% RSLogix 500 project LVD190607.RSS, saved by version 11.00.00.00 %
PROJECT "LINL0619"    % processor: MicroLogix 1400 %

PROGRAM FILES
  LAD 2 "MAIN"  60 rungs  % Main Program Routine %
  LAD 3 "TEST"  7 rungs
  LAD 4 "ENABLES"  16 rungs
  LAD 6 "FEED"  11 rungs  % normal %
  LAD 8 "SPEEDS"  12 rungs
  LAD 20 "HSC BOT"  5 rungs
  LAD 22 "HSC TOP"  5 rungs
  LAD 30 "1 MS STI"  23 rungs  % high speed %
  LAD 40 "SHIFT BOT"  8 rungs
  LAD 42 "SHIFT TOP"  10 rungs
  LAD 50 "BOTOPTIC"  3 rungs
  LAD 52 "BOTOPTMES"  7 rungs
  LAD 80 "XFER"  3 rungs
  LAD 90 "TOPOPTIC"  10 rungs
  LAD 91 "TOPOPVERT"  13 rungs
  LAD 92 "TOPOPREAL"  19 rungs
  LAD 93 "TOPOPTEST"  8 rungs
  LAD 94 "TOPOPRANGE"  6 rungs
  LAD 95 "TOPOPOKAY"  6 rungs
  LAD 96 "TESTINJECT"  10 rungs
  LAD 100 "I5"  22 rungs
  LAD 101 "I5 RESULT"  7 rungs
  LAD 102 "I5 PASS"  6 rungs
  LAD 103 "I5 FAIL"  4 rungs
  LAD 104 "I5 ACQ"  9 rungs
  LAD 105 "I5 TESTER"  5 rungs
  LAD 106 "I5 TRIG"  5 rungs
  LAD 107 "I5 FIFOSET"  9 rungs
  LAD 108 "I5 FIFOGET"  8 rungs
  LAD 109 "I5 DATA"  3 rungs
  LAD 110 "I5 FAULT"  9 rungs
  LAD 111 "I5 FIX1"  5 rungs
  LAD 112 "I5 FIX2"  3 rungs
  LAD 120 "I6"  21 rungs
  LAD 121 "I6 RESULT"  7 rungs
  LAD 122 "I6 PASS"  5 rungs
  LAD 123 "I6 FAIL"  3 rungs
  LAD 124 "I6 ACQ"  8 rungs
  LAD 125 "I6 TESTER"  5 rungs
  LAD 126 "I6 TRIG"  5 rungs
  LAD 127 "I6 FIFOSET"  9 rungs
  LAD 128 "I6 FIFOGET"  8 rungs
  LAD 129 "I6 DATA"  3 rungs
  LAD 130 "I6 FAULT"  9 rungs
  LAD 131 "I6 FIX1"  5 rungs
  LAD 132 "I6 FIX2"  3 rungs
  LAD 140 "I7"  21 rungs
  LAD 141 "I7 RESULT"  7 rungs
  LAD 142 "I7 PASS"  6 rungs
  LAD 143 "I7 FAIL"  4 rungs
  LAD 144 "I7 ACQ"  9 rungs
  LAD 145 "I7 TESTER"  5 rungs
  LAD 146 "I7 TRIG"  5 rungs
  LAD 147 "I7 FIFOSET"  9 rungs
  LAD 148 "I7 FIFOGET"  8 rungs
  LAD 149 "I7 DATA"  3 rungs
  LAD 150 "I7 FAULT"  9 rungs
  LAD 151 "I7 FIX1"  5 rungs
  LAD 152 "I7 FIX2"  3 rungs
  LAD 160 "I8"  22 rungs
  LAD 161 "I8 RESULT"  7 rungs
  LAD 162 "I8 PASS"  6 rungs
  LAD 163 "I8 FAIL"  4 rungs
  LAD 164 "I8 ACQ"  9 rungs
  LAD 165 "I8 TESTER"  5 rungs
  LAD 166 "I8 TRIG"  5 rungs
  LAD 167 "I8 FIFOSET"  9 rungs
  LAD 168 "I8 FIFOGET"  8 rungs
  LAD 169 "I8 DATA"  3 rungs
  LAD 170 "I8 FAULT"  9 rungs
  LAD 171 "I8 FIX1"  5 rungs
  LAD 172 "I8 FIX2"  3 rungs
  LAD 200 "PASS BLOW"  15 rungs
  LAD 213 "TESTTRIG1"  4 rungs
  LAD 214 "TESTTRIG5"  4 rungs
  LAD 215 "TESTTRIG6"  4 rungs
  LAD 216 "TESTTRIG7"  4 rungs
  LAD 217 "TESTTRIG8"  4 rungs
  LAD 219 "PACKAGER"  28 rungs  % normal %
  LAD 220 "NO PACKAGE"  8 rungs
  LAD 222 "RATE1"  9 rungs
  LAD 223 "RATE2"  6 rungs
  LAD 224 "RESET RATE"  6 rungs
  LAD 240 "NP STOP"  8 rungs
  LAD 246 "SPEED BOT"  8 rungs  % high speed %
  LAD 248 "SPEED TOP"  8 rungs  % high speed %
  LAD 250 "P BOT"  7 rungs  % high speed %
  LAD 252 "P TOP"  7 rungs  % high speed %
  LAD 254 "TOTALCOUNT"  4 rungs
  LAD 255 "SAVED"  4 rungs

DATA FILES
  O0 OUTPUT  11 elements
  I1 INPUT  11 elements
  S2 STATUS  66 elements
  B3 BINARY  14 elements
  T4 TIMER  45 elements
  C5 COUNTER  1 elements
  R6 CONTROL  30 elements
  N7 INTEGER  200 elements
  F8 FLOAT  100 elements
  B12 HMI_BINARY  22 elements  % general use with hmi to avoid additional reads %
  L13  COUNTS  256 elements
  F14 HMI_FLOATS  100 elements
  N15 HMI_INTS  100 elements
  L16 HMI_LONGS  100 elements
  L19 RATE DATA  50 elements
  L20 I7TIMEFIFO  50 elements
  L21 I7POSFIFO  50 elements
  L22 I8TIMEFIFO  50 elements
  L23 I8POSFIFO  50 elements
  L30 INS5TIME  50 elements
  L31 INS5POS  50 elements
  L32 INS6TIME  50 elements
  L33 INS6POS  50 elements
  B34 BOT NG  128 elements
  B35 TOP NG  128 elements
  B36 BOTGOOD  128 elements
  B37 TOPGOOD1  128 elements
  B38 EX1 TEST  128 elements
  B39 TOPGOOD2  128 elements
  B40 EX2 TEST  128 elements
  N184 TEST INTS  50 elements
  L192 SPD OFFSET  50 elements
  B196 CTRL BITS  50 elements
  L199 USED  36 elements

LADDER 2 "MAIN"    % Main Program Routine %
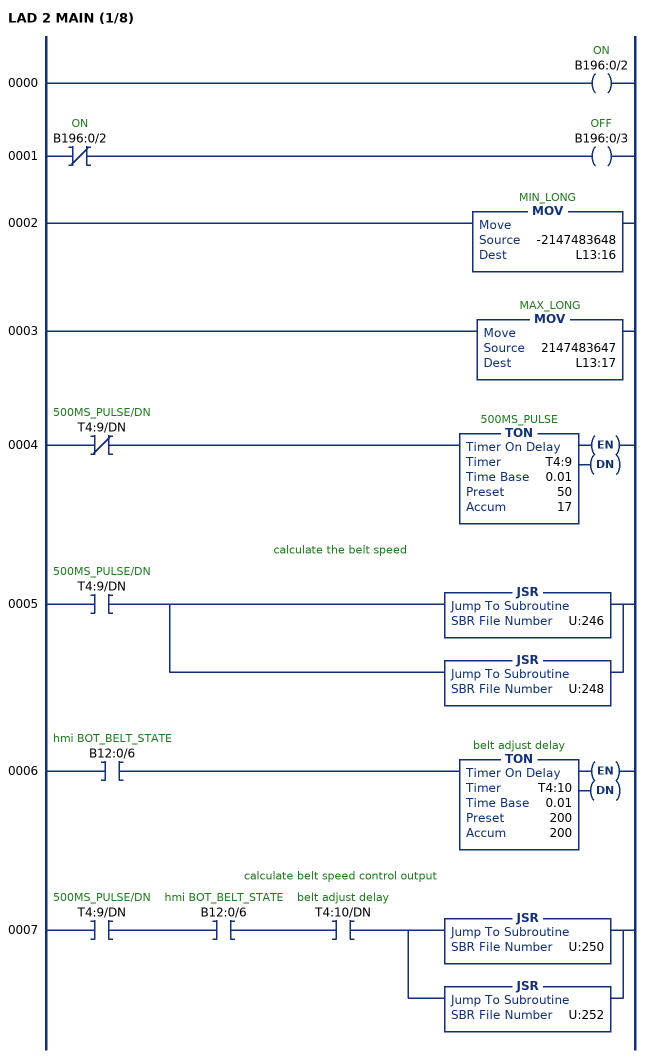
% Rung: 0 %
SOR OTE B196:0/2 EOR
%   B196:0/2  ON %
% Rung: 1 %
SOR XIO B196:0/2 OTE B196:0/3 EOR
%   B196:0/2  ON %
%   B196:0/3  OFF %
% Rung: 2 %
SOR MOV -2147483648 L13:16 EOR
%   L13:16  MIN_LONG %
% Rung: 3 %
SOR MOV 2147483647 L13:17 EOR
%   L13:17  MAX_LONG %
% Rung: 4 %
SOR XIO T4:9/DN TON T4:9 0.01 50 17 EOR
%   T4:9  500MS_PULSE %
% Rung: 5 %
% calculate the belt speed %
SOR XIC T4:9/DN BST JSR U:246 NXB JSR U:248 BND EOR
%   T4:9  500MS_PULSE %
% Rung: 6 %
SOR XIC B12:0/6 TON T4:10 0.01 200 200 EOR
%   B12:0/6  BOT_BELT_STATE  "hmi" %
%   T4:10  "belt adjust delay" %
% Rung: 7 %
% calculate belt speed control output %
SOR XIC T4:9/DN XIC B12:0/6 XIC T4:10/DN BST JSR U:250 NXB JSR U:252 BND EOR
%   T4:9  500MS_PULSE %
%   B12:0/6  BOT_BELT_STATE  "hmi" %
%   T4:10  "belt adjust delay" %

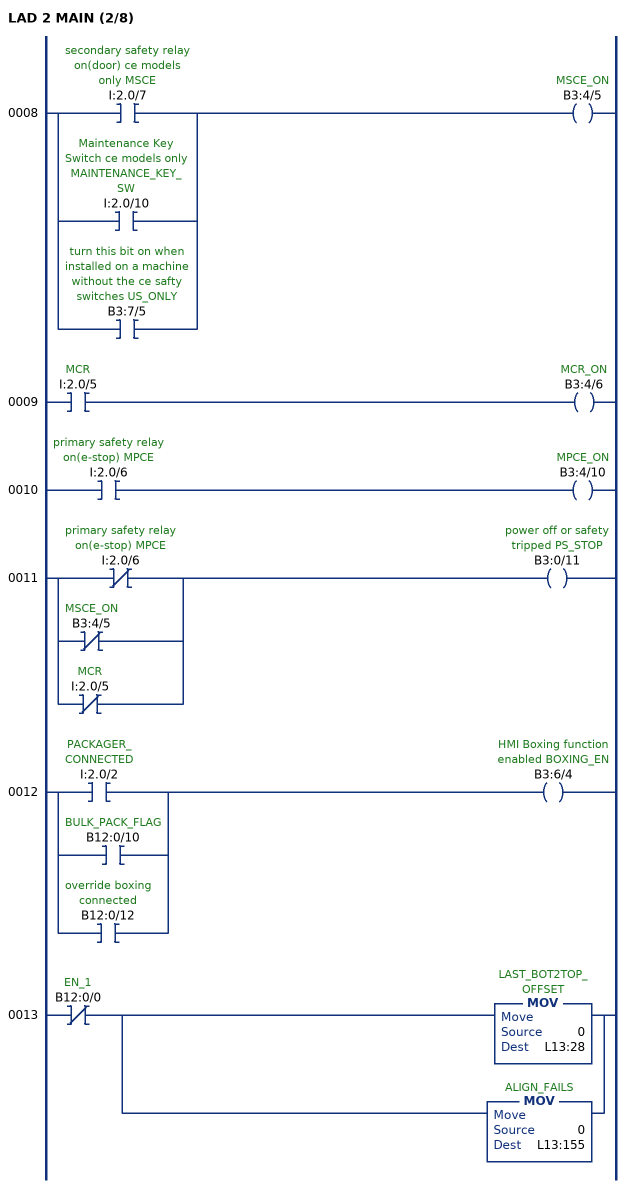
% Rung: 8 %
SOR BST XIC I:2.0/7 NXB XIC I:2.0/10 NXB XIC B3:7/5 BND OTE B3:4/5 EOR
%   I:2.0/7  MSCE  "secondary safety relay on(door) ce models only" %
%   I:2.0/10  MAINTENANCE_KEY_SW  "Maintenance Key Switch ce models only" %
%   B3:7/5  US_ONLY  "turn this bit on when installed on a machine without the ce safty switches" %
%   B3:4/5  MSCE_ON %
% Rung: 9 %
SOR XIC I:2.0/5 OTE B3:4/6 EOR
%   I:2.0/5  MCR %
%   B3:4/6  MCR_ON %
% Rung: 10 %
SOR XIC I:2.0/6 OTE B3:4/10 EOR
%   I:2.0/6  MPCE  "primary safety relay on(e-stop)" %
%   B3:4/10  MPCE_ON %
% Rung: 11 %
SOR BST XIO I:2.0/6 NXB XIO B3:4/5 NXB XIO I:2.0/5 BND OTE B3:0/11 EOR
%   I:2.0/6  MPCE  "primary safety relay on(e-stop)" %
%   B3:4/5  MSCE_ON %
%   I:2.0/5  MCR %
%   B3:0/11  PS_STOP  "power off or safety tripped" %
% Rung: 12 %
SOR BST XIC I:2.0/2 NXB XIC B12:0/10 NXB XIC B12:0/12 BND OTE B3:6/4 EOR
%   I:2.0/2  PACKAGER_CONNECTED %
%   B12:0/10  BULK_PACK_FLAG %
%   B12:0/12  "override boxing connected" %
%   B3:6/4  BOXING_EN  "HMI Boxing function enabled" %
% Rung: 13 %
SOR XIO B12:0/0 BST MOV 0 L13:28 NXB MOV 0 L13:155 BND EOR
%   B12:0/0  EN_1 %
%   L13:28  LAST_BOT2TOP_OFFSET %
%   L13:155  ALIGN_FAILS %

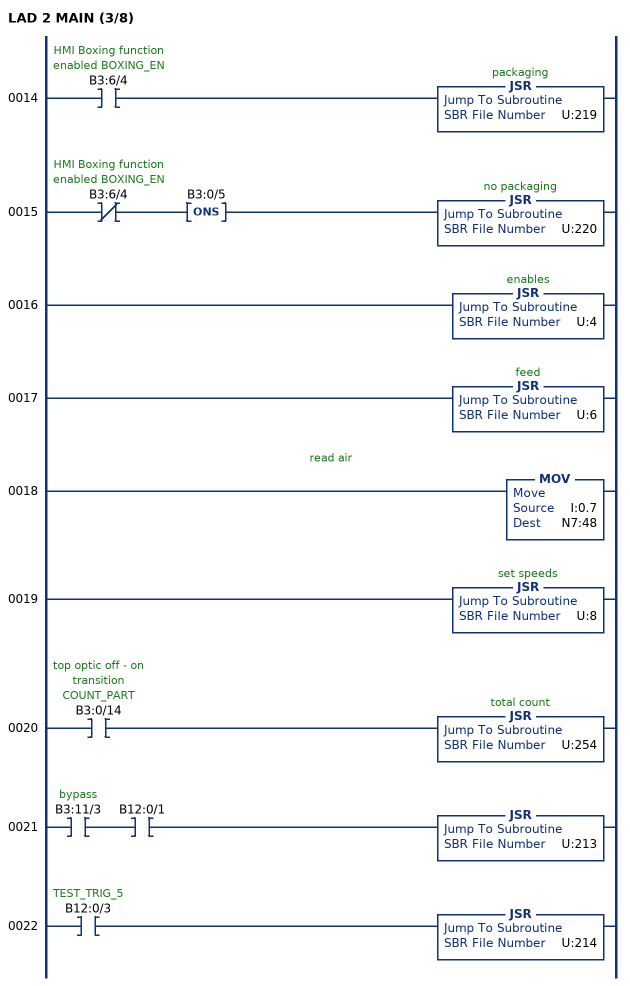
% Rung: 14 %
SOR XIC B3:6/4 JSR U:219 EOR
%   B3:6/4  BOXING_EN  "HMI Boxing function enabled" %
%   U:219  "packaging" %
% Rung: 15 %
SOR XIO B3:6/4 ONS B3:0/5 JSR U:220 EOR
%   B3:6/4  BOXING_EN  "HMI Boxing function enabled" %
%   U:220  "no packaging" %
% Rung: 16 %
SOR JSR U:4 EOR
%   U:4  "enables" %
% Rung: 17 %
SOR JSR U:6 EOR
%   U:6  "feed" %
% Rung: 18 %
% read air %
SOR MOV I:0.7 N7:48 EOR
%   I:0.7  "Air Presure Sensor Input Signal" %
% Rung: 19 %
SOR JSR U:8 EOR
%   U:8  "set speeds" %
% Rung: 20 %
SOR XIC B3:0/14 JSR U:254 EOR
%   B3:0/14  COUNT_PART  "top optic off - on transition" %
%   U:254  "total count" %
% Rung: 21 %
SOR XIC B3:11/3 XIC B12:0/1 JSR U:213 EOR
%   B3:11/3  "bypass" %
% Rung: 22 %
SOR XIC B12:0/3 JSR U:214 EOR
%   B12:0/3  TEST_TRIG_5 %

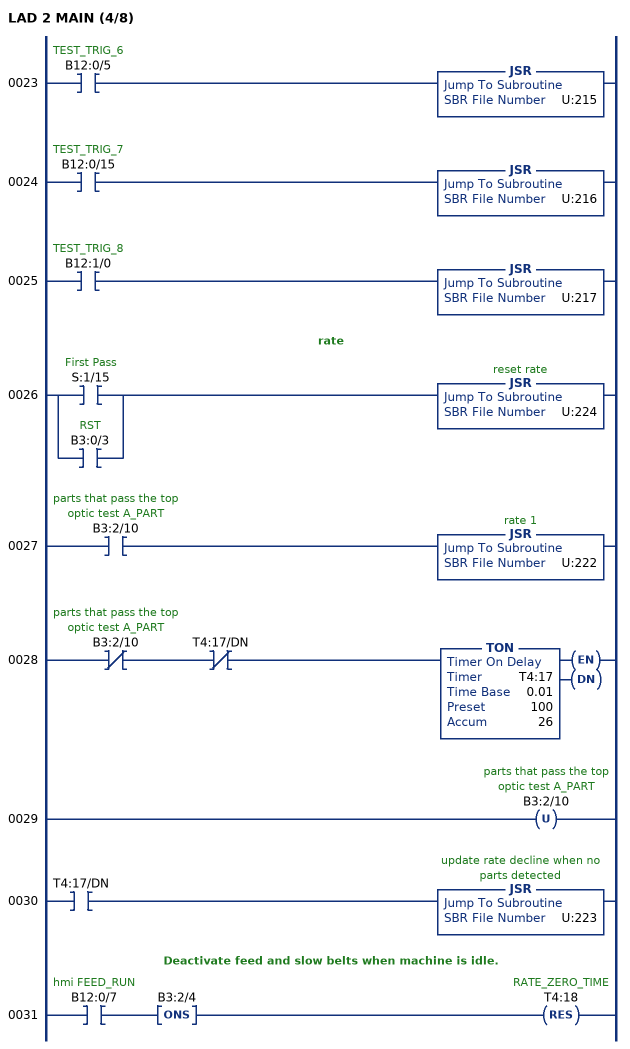
% Rung: 23 %
SOR XIC B12:0/5 JSR U:215 EOR
%   B12:0/5  TEST_TRIG_6 %
% Rung: 24 %
SOR XIC B12:0/15 JSR U:216 EOR
%   B12:0/15  TEST_TRIG_7 %
% Rung: 25 %
SOR XIC B12:1/0 JSR U:217 EOR
%   B12:1/0  TEST_TRIG_8 %
% Rung: 26 %
% TITLE: rate %
SOR BST XIC S:1/15 NXB XIC B3:0/3 BND JSR U:224 EOR
%   S:1/15  "First Pass" %
%   B3:0/3  RST %
%   U:224  "reset rate" %
% Rung: 27 %
SOR XIC B3:2/10 JSR U:222 EOR
%   B3:2/10  A_PART  "parts that pass the top optic test" %
%   U:222  "rate 1" %
% Rung: 28 %
SOR XIO B3:2/10 XIO T4:17/DN TON T4:17 0.01 100 26 EOR
%   B3:2/10  A_PART  "parts that pass the top optic test" %
% Rung: 29 %
SOR OTU B3:2/10 EOR
%   B3:2/10  A_PART  "parts that pass the top optic test" %
% Rung: 30 %
SOR XIC T4:17/DN JSR U:223 EOR
%   U:223  "update rate decline when no parts detected" %
% Rung: 31 %
% TITLE: Deactivate feed and slow belts when machine is idle. %
SOR XIC B12:0/7 ONS B3:2/4 RES T4:18 EOR
%   B12:0/7  FEED_RUN  "hmi" %
%   T4:18  RATE_ZERO_TIME %

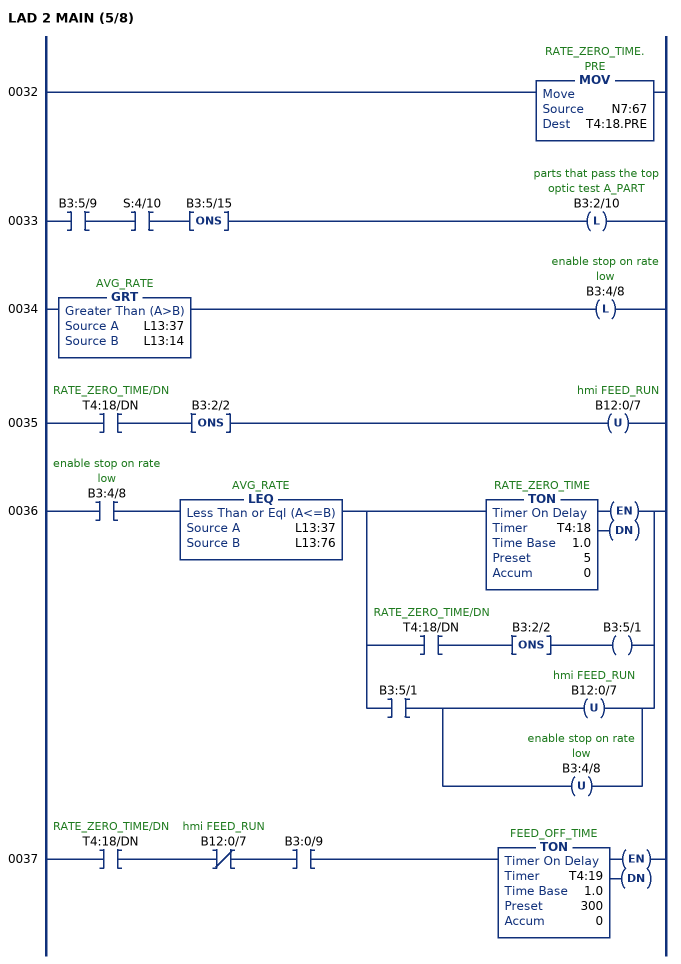
% Rung: 32 %
SOR MOV N7:67 T4:18.PRE EOR
%   N7:67  "empty bowl or jam bowl run time" %
%   T4:18  RATE_ZERO_TIME %
% Rung: 33 %
SOR XIC B3:5/9 XIC S:4/10 ONS B3:5/15 OTL B3:2/10 EOR
%   B3:2/10  A_PART  "parts that pass the top optic test" %
% Rung: 34 %
SOR GRT L13:37 L13:14 OTL B3:4/8 EOR
%   L13:37  AVG_RATE %
%   B3:4/8  "enable stop on rate low" %
% Rung: 35 %
SOR XIC T4:18/DN ONS B3:2/2 OTU B12:0/7 EOR
%   T4:18  RATE_ZERO_TIME %
%   B12:0/7  FEED_RUN  "hmi" %
% Rung: 36 %
SOR XIC B3:4/8 LEQ L13:37 L13:76 BST TON T4:18 1.0 5 0 NXB XIC T4:18/DN ONS B3:2/2 OTE B3:5/1 NXB XIC B3:5/1 BST OTU B12:0/7 NXB OTU B3:4/8 BND BND EOR
%   B3:4/8  "enable stop on rate low" %
%   L13:37  AVG_RATE %
%   T4:18  RATE_ZERO_TIME %
%   B12:0/7  FEED_RUN  "hmi" %
% Rung: 37 %
SOR XIC T4:18/DN XIO B12:0/7 XIC B3:0/9 TON T4:19 1.0 300 0 EOR
%   T4:18  RATE_ZERO_TIME %
%   B12:0/7  FEED_RUN  "hmi" %
%   T4:19  FEED_OFF_TIME %

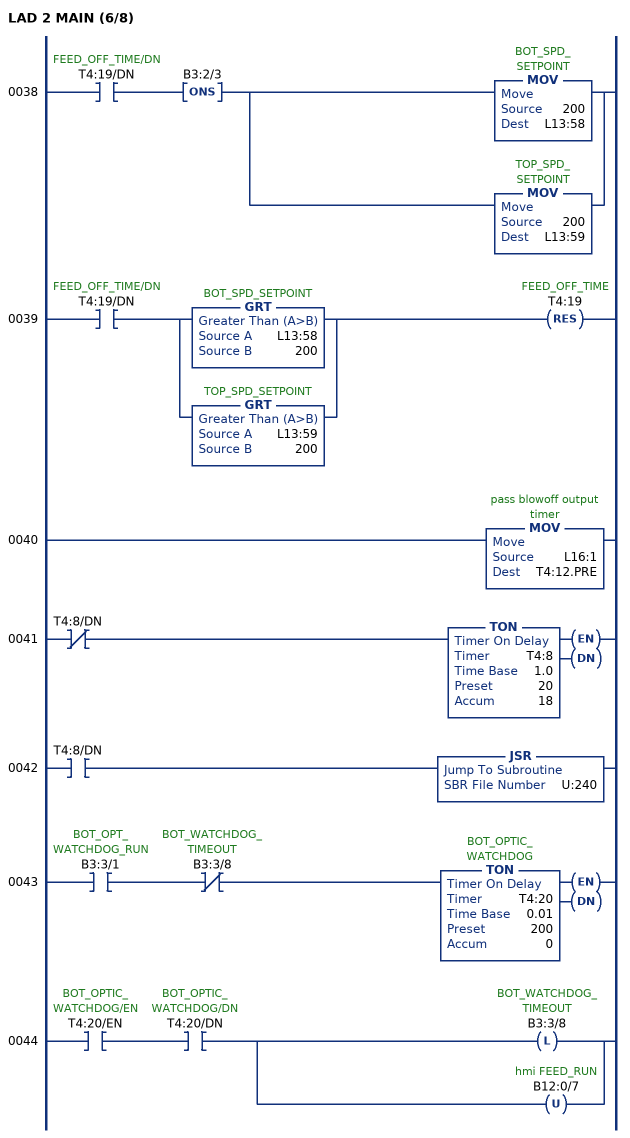
% Rung: 38 %
SOR XIC T4:19/DN ONS B3:2/3 BST MOV 200 L13:58 NXB MOV 200 L13:59 BND EOR
%   T4:19  FEED_OFF_TIME %
%   L13:58  BOT_SPD_SETPOINT %
%   L13:59  TOP_SPD_SETPOINT %
% Rung: 39 %
SOR XIC T4:19/DN BST GRT L13:58 200 NXB GRT L13:59 200 BND RES T4:19 EOR
%   T4:19  FEED_OFF_TIME %
%   L13:58  BOT_SPD_SETPOINT %
%   L13:59  TOP_SPD_SETPOINT %
% Rung: 40 %
SOR MOV L16:1 T4:12.PRE EOR
%   L16:1  BLOW_TIME %
%   T4:12  "pass blowoff output timer" %
% Rung: 41 %
SOR XIO T4:8/DN TON T4:8 1.0 20 18 EOR
% Rung: 42 %
SOR XIC T4:8/DN JSR U:240 EOR
% Rung: 43 %
SOR XIC B3:3/1 XIO B3:3/8 TON T4:20 0.01 200 0 EOR
%   B3:3/1  BOT_OPT_WATCHDOG_RUN %
%   B3:3/8  BOT_WATCHDOG_TIMEOUT %
%   T4:20  BOT_OPTIC_WATCHDOG %
% Rung: 44 %
SOR XIC T4:20/EN XIC T4:20/DN BST OTL B3:3/8 NXB OTU B12:0/7 BND EOR
%   T4:20  BOT_OPTIC_WATCHDOG %
%   B3:3/8  BOT_WATCHDOG_TIMEOUT %
%   B12:0/7  FEED_RUN  "hmi" %

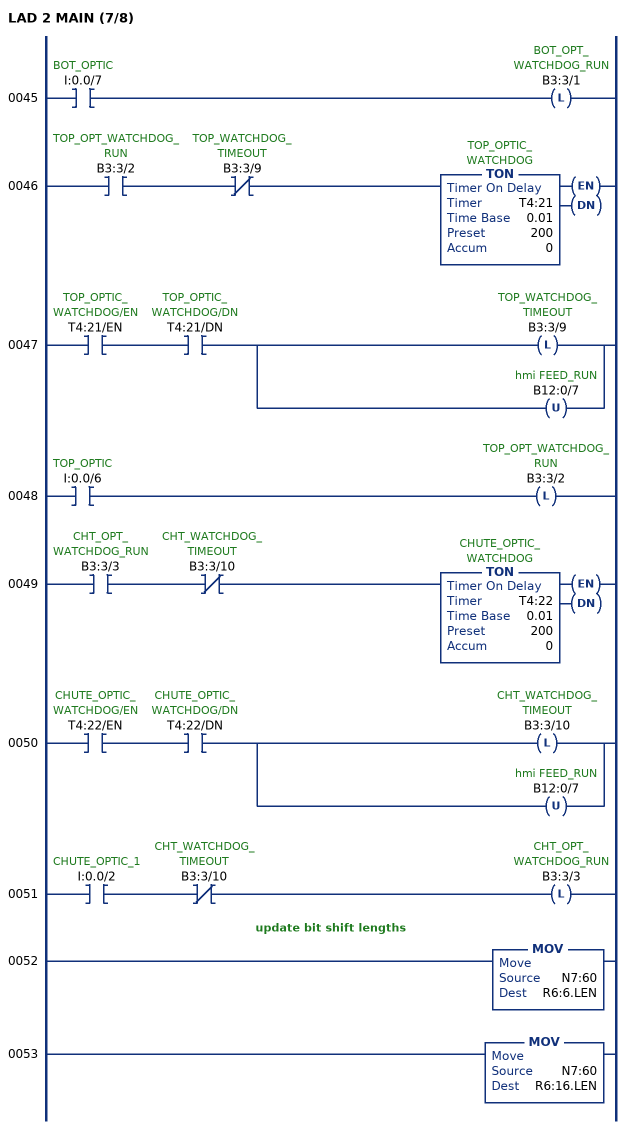
% Rung: 45 %
SOR XIC I:0.0/7 OTL B3:3/1 EOR
%   I:0.0/7  BOT_OPTIC %
%   B3:3/1  BOT_OPT_WATCHDOG_RUN %
% Rung: 46 %
SOR XIC B3:3/2 XIO B3:3/9 TON T4:21 0.01 200 0 EOR
%   B3:3/2  TOP_OPT_WATCHDOG_RUN %
%   B3:3/9  TOP_WATCHDOG_TIMEOUT %
%   T4:21  TOP_OPTIC_WATCHDOG %
% Rung: 47 %
SOR XIC T4:21/EN XIC T4:21/DN BST OTL B3:3/9 NXB OTU B12:0/7 BND EOR
%   T4:21  TOP_OPTIC_WATCHDOG %
%   B3:3/9  TOP_WATCHDOG_TIMEOUT %
%   B12:0/7  FEED_RUN  "hmi" %
% Rung: 48 %
SOR XIC I:0.0/6 OTL B3:3/2 EOR
%   I:0.0/6  TOP_OPTIC %
%   B3:3/2  TOP_OPT_WATCHDOG_RUN %
% Rung: 49 %
SOR XIC B3:3/3 XIO B3:3/10 TON T4:22 0.01 200 0 EOR
%   B3:3/3  CHT_OPT_WATCHDOG_RUN %
%   B3:3/10  CHT_WATCHDOG_TIMEOUT %
%   T4:22  CHUTE_OPTIC_WATCHDOG %
% Rung: 50 %
SOR XIC T4:22/EN XIC T4:22/DN BST OTL B3:3/10 NXB OTU B12:0/7 BND EOR
%   T4:22  CHUTE_OPTIC_WATCHDOG %
%   B3:3/10  CHT_WATCHDOG_TIMEOUT %
%   B12:0/7  FEED_RUN  "hmi" %
% Rung: 51 %
SOR XIC I:0.0/2 XIO B3:3/10 OTL B3:3/3 EOR
%   I:0.0/2  CHUTE_OPTIC_1 %
%   B3:3/10  CHT_WATCHDOG_TIMEOUT %
%   B3:3/3  CHT_OPT_WATCHDOG_RUN %
% Rung: 52 %
% TITLE: update bit shift lengths %
SOR MOV N7:60 R6:6.LEN EOR
% Rung: 53 %
SOR MOV N7:60 R6:16.LEN EOR

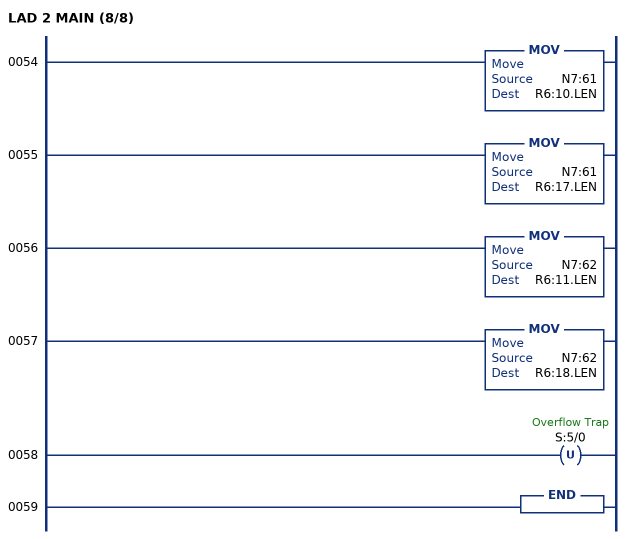
% Rung: 54 %
SOR MOV N7:61 R6:10.LEN EOR
% Rung: 55 %
SOR MOV N7:61 R6:17.LEN EOR
% Rung: 56 %
SOR MOV N7:62 R6:11.LEN EOR
% Rung: 57 %
SOR MOV N7:62 R6:18.LEN EOR
% Rung: 58 %
SOR OTU S:5/0 EOR
%   S:5/0  "Overflow Trap" %
% Rung: 59 %
SOR END EOR

LADDER 3 "TEST"
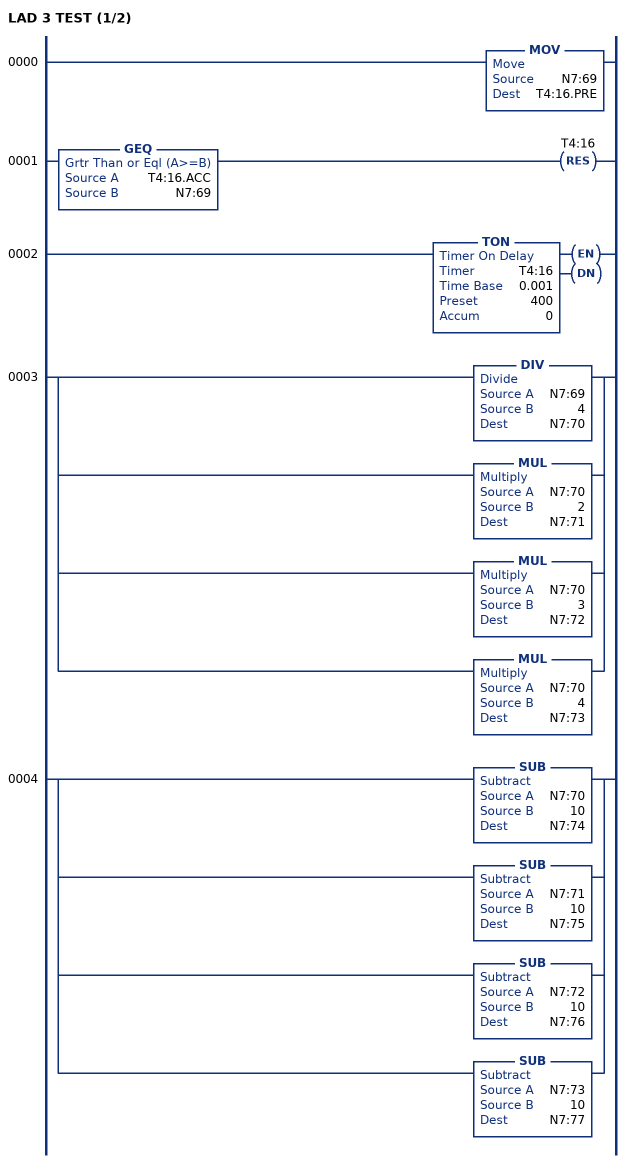
% Rung: 0 %
SOR MOV N7:69 T4:16.PRE EOR
% Rung: 1 %
SOR GEQ T4:16.ACC N7:69 RES T4:16 EOR
% Rung: 2 %
SOR TON T4:16 0.001 400 0 EOR
% Rung: 3 %
SOR BST DIV N7:69 4 N7:70 NXB MUL N7:70 2 N7:71 NXB MUL N7:70 3 N7:72 NXB MUL N7:70 4 N7:73 BND EOR
% Rung: 4 %
SOR BST SUB N7:70 10 N7:74 NXB SUB N7:71 10 N7:75 NXB SUB N7:72 10 N7:76 NXB SUB N7:73 10 N7:77 BND EOR

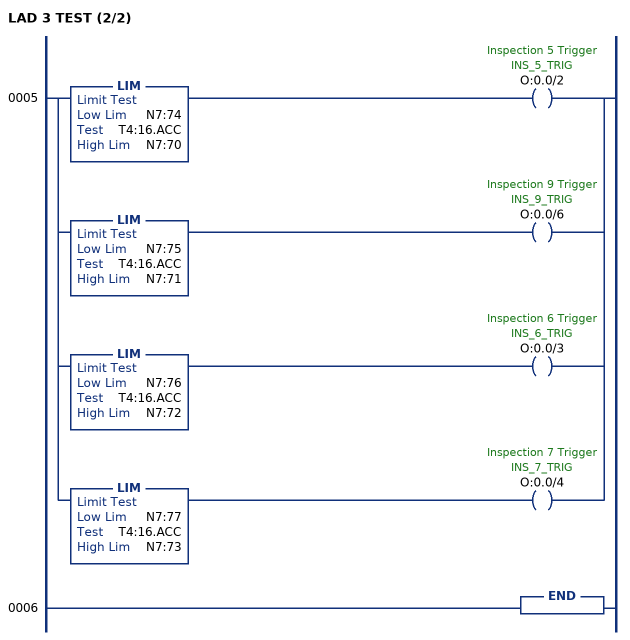
% Rung: 5 %
SOR BST LIM N7:74 T4:16.ACC N7:70 OTE O:0.0/2 NXB LIM N7:75 T4:16.ACC N7:71 OTE O:0.0/6 NXB LIM N7:76 T4:16.ACC N7:72 OTE O:0.0/3 NXB LIM N7:77 T4:16.ACC N7:73 OTE O:0.0/4 BND EOR
%   O:0.0/2  INS_5_TRIG  "Inspection 5 Trigger" %
%   O:0.0/6  INS_9_TRIG  "Inspection 9 Trigger" %
%   O:0.0/3  INS_6_TRIG  "Inspection 6 Trigger" %
%   O:0.0/4  INS_7_TRIG  "Inspection 7 Trigger" %
% Rung: 6 %
SOR END EOR

LADDER 4 "ENABLES"
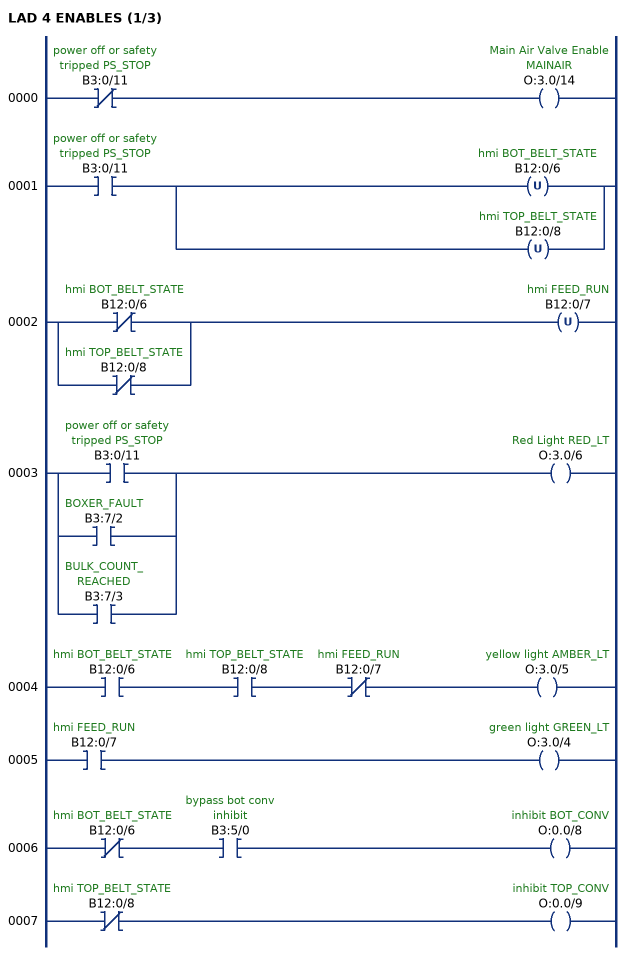
% Rung: 0 %
SOR XIO B3:0/11 OTE O:3.0/14 EOR
%   B3:0/11  PS_STOP  "power off or safety tripped" %
%   O:3.0/14  MAINAIR  "Main Air Valve Enable" %
% Rung: 1 %
SOR XIC B3:0/11 BST OTU B12:0/6 NXB OTU B12:0/8 BND EOR
%   B3:0/11  PS_STOP  "power off or safety tripped" %
%   B12:0/6  BOT_BELT_STATE  "hmi" %
%   B12:0/8  TOP_BELT_STATE  "hmi" %
% Rung: 2 %
SOR BST XIO B12:0/6 NXB XIO B12:0/8 BND OTU B12:0/7 EOR
%   B12:0/6  BOT_BELT_STATE  "hmi" %
%   B12:0/8  TOP_BELT_STATE  "hmi" %
%   B12:0/7  FEED_RUN  "hmi" %
% Rung: 3 %
SOR BST XIC B3:0/11 NXB XIC B3:7/2 NXB XIC B3:7/3 BND OTE O:3.0/6 EOR
%   B3:0/11  PS_STOP  "power off or safety tripped" %
%   B3:7/2  BOXER_FAULT %
%   B3:7/3  BULK_COUNT_REACHED %
%   O:3.0/6  RED_LT  "Red Light" %
% Rung: 4 %
SOR XIC B12:0/6 XIC B12:0/8 XIO B12:0/7 OTE O:3.0/5 EOR
%   B12:0/6  BOT_BELT_STATE  "hmi" %
%   B12:0/8  TOP_BELT_STATE  "hmi" %
%   B12:0/7  FEED_RUN  "hmi" %
%   O:3.0/5  AMBER_LT  "yellow light" %
% Rung: 5 %
SOR XIC B12:0/7 OTE O:3.0/4 EOR
%   B12:0/7  FEED_RUN  "hmi" %
%   O:3.0/4  GREEN_LT  "green light" %
% Rung: 6 %
SOR XIO B12:0/6 XIC B3:5/0 OTE O:0.0/8 EOR
%   B12:0/6  BOT_BELT_STATE  "hmi" %
%   B3:5/0  "bypass bot conv inhibit" %
%   O:0.0/8  BOT_CONV  "inhibit" %
% Rung: 7 %
SOR XIO B12:0/8 OTE O:0.0/9 EOR
%   B12:0/8  TOP_BELT_STATE  "hmi" %
%   O:0.0/9  TOP_CONV  "inhibit" %

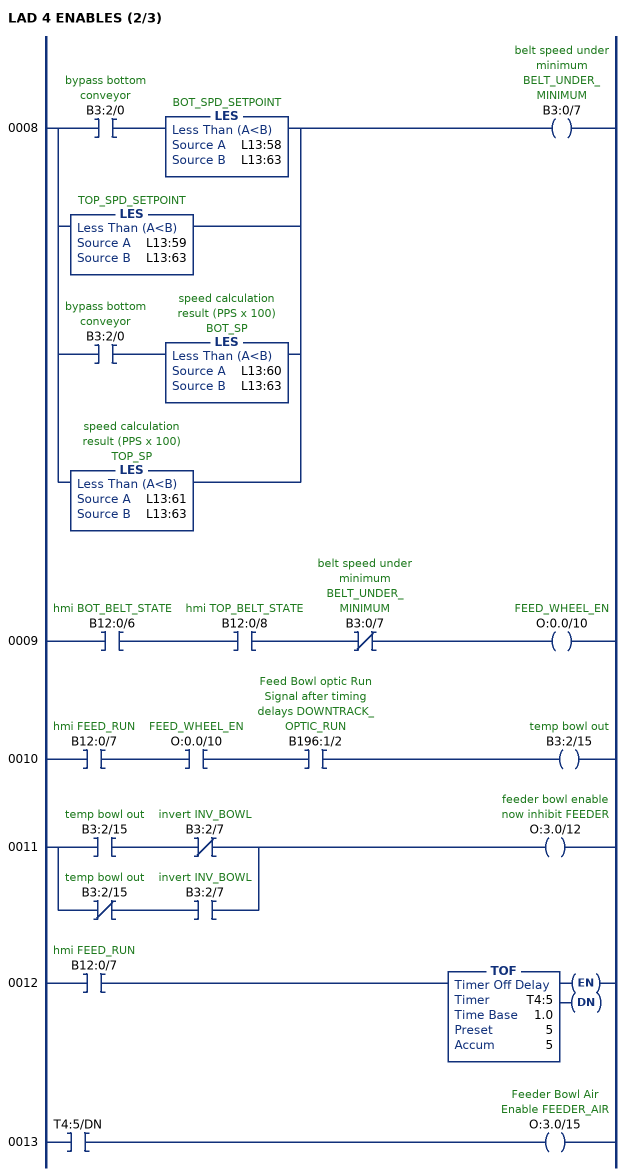
% Rung: 8 %
SOR BST XIC B3:2/0 LES L13:58 L13:63 NXB LES L13:59 L13:63 NXB XIC B3:2/0 LES L13:60 L13:63 NXB LES L13:61 L13:63 BND OTE B3:0/7 EOR
%   B3:2/0  "bypass bottom conveyor" %
%   L13:58  BOT_SPD_SETPOINT %
%   L13:63  "min belt speed" %
%   L13:59  TOP_SPD_SETPOINT %
%   L13:60  BOT_SP  "speed calculation result (PPS x 100)" %
%   L13:61  TOP_SP  "speed calculation result (PPS x 100)" %
%   B3:0/7  BELT_UNDER_MINIMUM  "belt speed under minimum" %
% Rung: 9 %
SOR XIC B12:0/6 XIC B12:0/8 XIO B3:0/7 OTE O:0.0/10 EOR
%   B12:0/6  BOT_BELT_STATE  "hmi" %
%   B12:0/8  TOP_BELT_STATE  "hmi" %
%   B3:0/7  BELT_UNDER_MINIMUM  "belt speed under minimum" %
%   O:0.0/10  FEED_WHEEL_EN %
% Rung: 10 %
SOR XIC B12:0/7 XIC O:0.0/10 XIC B196:1/2 OTE B3:2/15 EOR
%   B12:0/7  FEED_RUN  "hmi" %
%   O:0.0/10  FEED_WHEEL_EN %
%   B196:1/2  DOWNTRACK_OPTIC_RUN  "Feed Bowl optic Run Signal after timing delays" %
%   B3:2/15  "temp bowl out" %
% Rung: 11 %
SOR BST XIC B3:2/15 XIO B3:2/7 NXB XIO B3:2/15 XIC B3:2/7 BND OTE O:3.0/12 EOR
%   B3:2/15  "temp bowl out" %
%   B3:2/7  INV_BOWL  "invert" %
%   O:3.0/12  FEEDER  "feeder bowl enable now inhibit" %
% Rung: 12 %
SOR XIC B12:0/7 TOF T4:5 1.0 5 5 EOR
%   B12:0/7  FEED_RUN  "hmi" %
% Rung: 13 %
SOR XIC T4:5/DN OTE O:3.0/15 EOR
%   O:3.0/15  FEEDER_AIR  "Feeder Bowl Air Enable" %

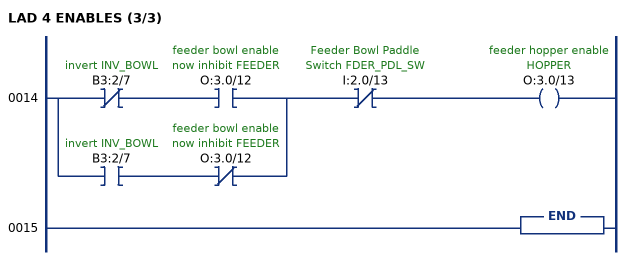
% Rung: 14 %
SOR BST XIO B3:2/7 XIC O:3.0/12 NXB XIC B3:2/7 XIO O:3.0/12 BND XIO I:2.0/13 OTE O:3.0/13 EOR
%   B3:2/7  INV_BOWL  "invert" %
%   O:3.0/12  FEEDER  "feeder bowl enable now inhibit" %
%   I:2.0/13  FDER_PDL_SW  "Feeder Bowl Paddle Switch" %
%   O:3.0/13  HOPPER  "feeder hopper enable" %
% Rung: 15 %
SOR END EOR

LADDER 6 "FEED"    % normal %
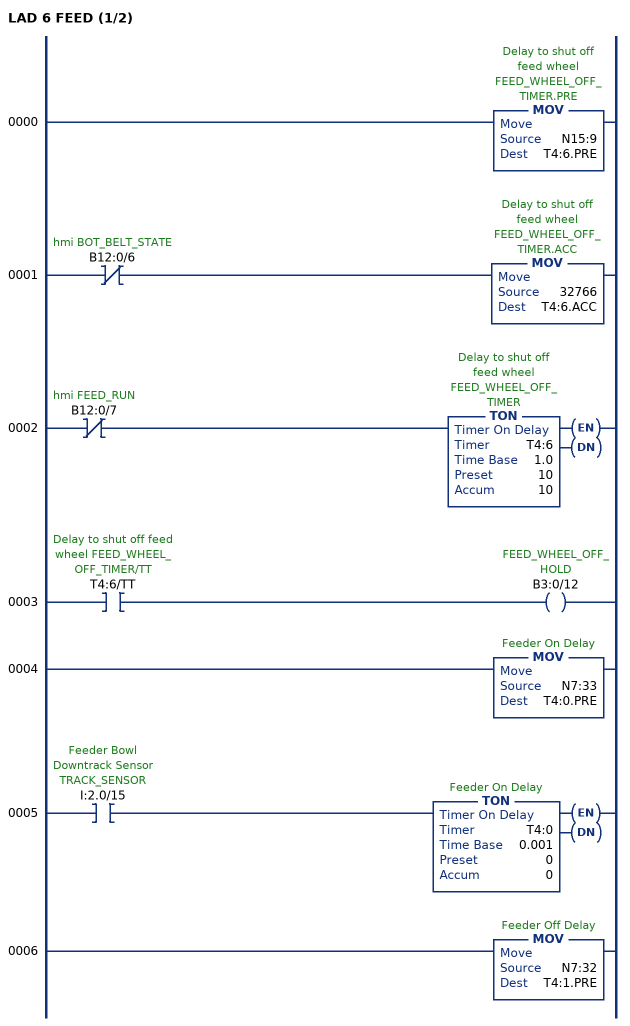
% Rung: 0 %
SOR MOV N15:9 T4:6.PRE EOR
%   N15:9  FEED_WHEEL_STOP_TIME %
%   T4:6  FEED_WHEEL_OFF_TIMER  "Delay to shut off feed wheel" %
% Rung: 1 %
SOR XIO B12:0/6 MOV 32766 T4:6.ACC EOR
%   B12:0/6  BOT_BELT_STATE  "hmi" %
%   T4:6  FEED_WHEEL_OFF_TIMER  "Delay to shut off feed wheel" %
% Rung: 2 %
SOR XIO B12:0/7 TON T4:6 1.0 10 10 EOR
%   B12:0/7  FEED_RUN  "hmi" %
%   T4:6  FEED_WHEEL_OFF_TIMER  "Delay to shut off feed wheel" %
% Rung: 3 %
SOR XIC T4:6/TT OTE B3:0/12 EOR
%   T4:6  FEED_WHEEL_OFF_TIMER  "Delay to shut off feed wheel" %
%   B3:0/12  FEED_WHEEL_OFF_HOLD %
% Rung: 4 %
SOR MOV N7:33 T4:0.PRE EOR
%   N7:33  "down track on delay" %
%   T4:0  "Feeder On Delay" %
% Rung: 5 %
SOR XIC I:2.0/15 TON T4:0 0.001 0 0 EOR
%   I:2.0/15  TRACK_SENSOR  "Feeder Bowl Downtrack Sensor" %
%   T4:0  "Feeder On Delay" %
% Rung: 6 %
SOR MOV N7:32 T4:1.PRE EOR
%   N7:32  "down track off delay" %
%   T4:1  "Feeder Off Delay" %

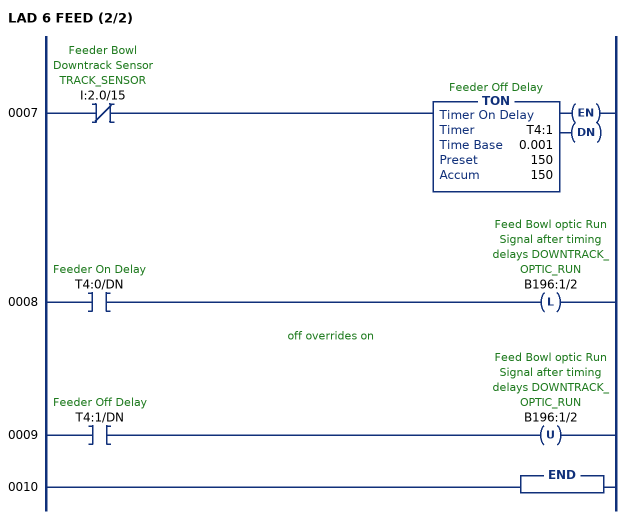
% Rung: 7 %
SOR XIO I:2.0/15 TON T4:1 0.001 150 150 EOR
%   I:2.0/15  TRACK_SENSOR  "Feeder Bowl Downtrack Sensor" %
%   T4:1  "Feeder Off Delay" %
% Rung: 8 %
SOR XIC T4:0/DN OTL B196:1/2 EOR
%   T4:0  "Feeder On Delay" %
%   B196:1/2  DOWNTRACK_OPTIC_RUN  "Feed Bowl optic Run Signal after timing delays" %
% Rung: 9 %
% off overrides on %
SOR XIC T4:1/DN OTU B196:1/2 EOR
%   T4:1  "Feeder Off Delay" %
%   B196:1/2  DOWNTRACK_OPTIC_RUN  "Feed Bowl optic Run Signal after timing delays" %
% Rung: 10 %
SOR END EOR

LADDER 8 "SPEEDS"
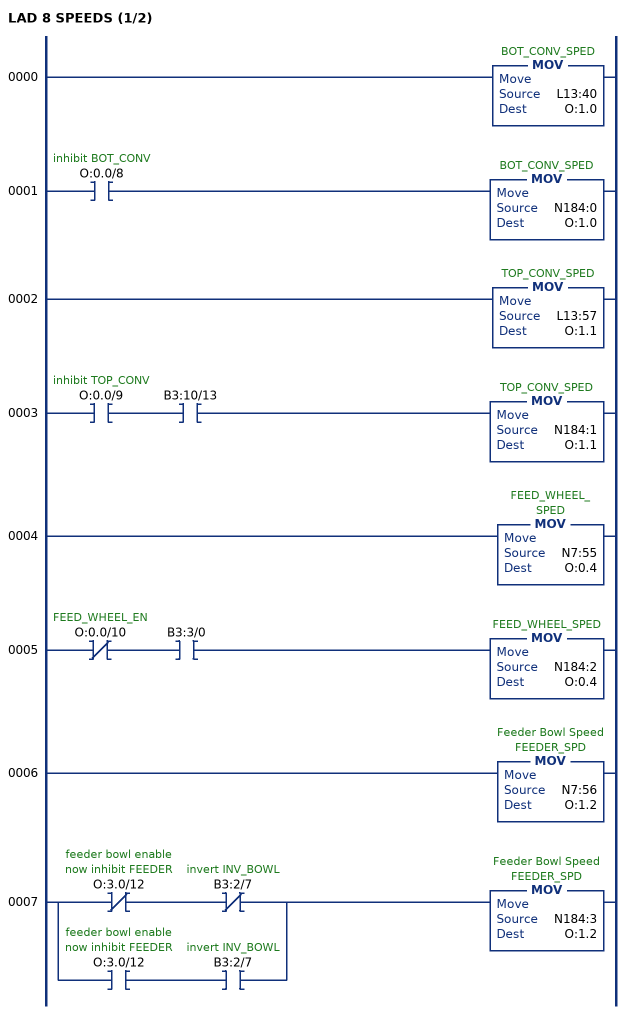
% Rung: 0 %
SOR MOV L13:40 O:1.0 EOR
%   L13:40  SCALED_BOT_VALUE %
%   O:1.0  BOT_CONV_SPED %
% Rung: 1 %
SOR XIC O:0.0/8 MOV N184:0 O:1.0 EOR
%   O:0.0/8  BOT_CONV  "inhibit" %
%   O:1.0  BOT_CONV_SPED %
% Rung: 2 %
SOR MOV L13:57 O:1.1 EOR
%   L13:57  SCALED_TOP_VALUE %
%   O:1.1  TOP_CONV_SPED %
% Rung: 3 %
SOR XIC O:0.0/9 XIC B3:10/13 MOV N184:1 O:1.1 EOR
%   O:0.0/9  TOP_CONV  "inhibit" %
%   O:1.1  TOP_CONV_SPED %
% Rung: 4 %
SOR MOV N7:55 O:0.4 EOR
%   O:0.4  FEED_WHEEL_SPED %
% Rung: 5 %
SOR XIO O:0.0/10 XIC B3:3/0 MOV N184:2 O:0.4 EOR
%   O:0.0/10  FEED_WHEEL_EN %
%   O:0.4  FEED_WHEEL_SPED %
% Rung: 6 %
SOR MOV N7:56 O:1.2 EOR
%   O:1.2  FEEDER_SPD  "Feeder Bowl Speed" %
% Rung: 7 %
SOR BST XIO O:3.0/12 XIO B3:2/7 NXB XIC O:3.0/12 XIC B3:2/7 BND MOV N184:3 O:1.2 EOR
%   O:3.0/12  FEEDER  "feeder bowl enable now inhibit" %
%   B3:2/7  INV_BOWL  "invert" %
%   O:1.2  FEEDER_SPD  "Feeder Bowl Speed" %

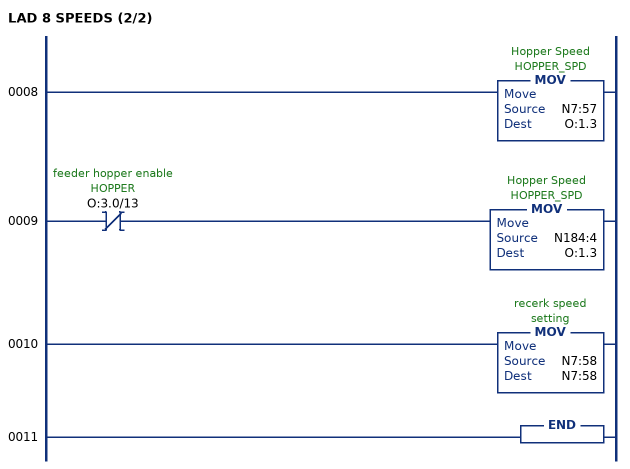
% Rung: 8 %
SOR MOV N7:57 O:1.3 EOR
%   O:1.3  HOPPER_SPD  "Hopper Speed" %
% Rung: 9 %
SOR XIO O:3.0/13 MOV N184:4 O:1.3 EOR
%   O:3.0/13  HOPPER  "feeder hopper enable" %
%   O:1.3  HOPPER_SPD  "Hopper Speed" %
% Rung: 10 %
SOR MOV N7:58 N7:58 EOR
%   N7:58  "recerk speed setting" %
% Rung: 11 %
SOR END EOR

LADDER 20 "HSC BOT"
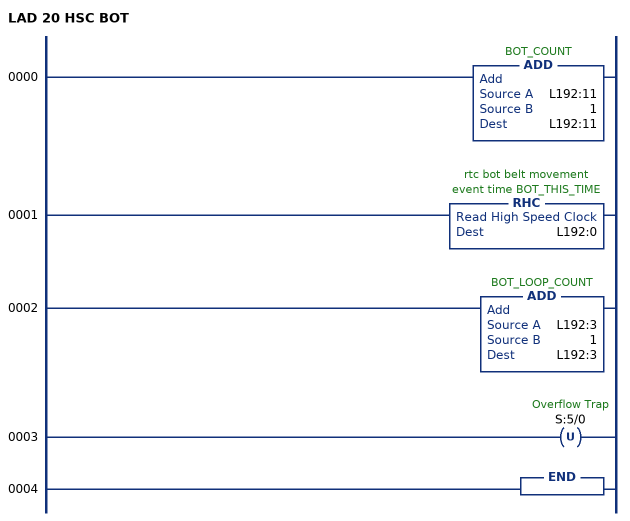
% Rung: 0 %
SOR ADD L192:11 1 L192:11 EOR
%   L192:11  BOT_COUNT %
% Rung: 1 %
SOR RHC L192:0 EOR
%   L192:0  BOT_THIS_TIME  "rtc bot belt movement event time" %
% Rung: 2 %
SOR ADD L192:3 1 L192:3 EOR
%   L192:3  BOT_LOOP_COUNT %
% Rung: 3 %
SOR OTU S:5/0 EOR
%   S:5/0  "Overflow Trap" %
% Rung: 4 %
SOR END EOR

LADDER 22 "HSC TOP"
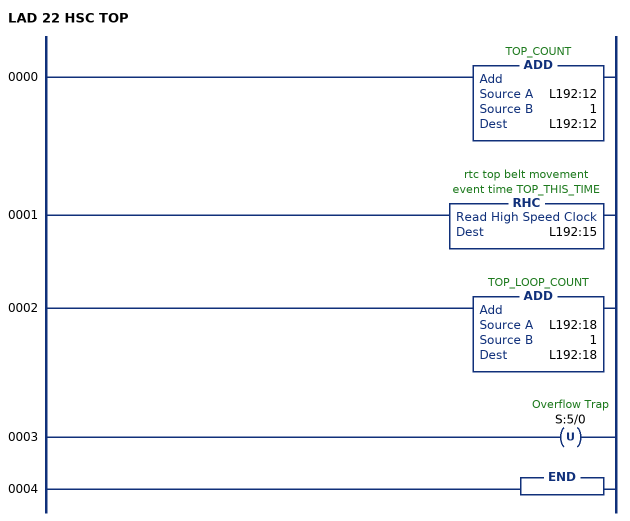
% Rung: 0 %
SOR ADD L192:12 1 L192:12 EOR
%   L192:12  TOP_COUNT %
% Rung: 1 %
SOR RHC L192:15 EOR
%   L192:15  TOP_THIS_TIME  "rtc top belt movement event time" %
% Rung: 2 %
SOR ADD L192:18 1 L192:18 EOR
%   L192:18  TOP_LOOP_COUNT %
% Rung: 3 %
SOR OTU S:5/0 EOR
%   S:5/0  "Overflow Trap" %
% Rung: 4 %
SOR END EOR

LADDER 30 "1 MS STI"    % high speed %
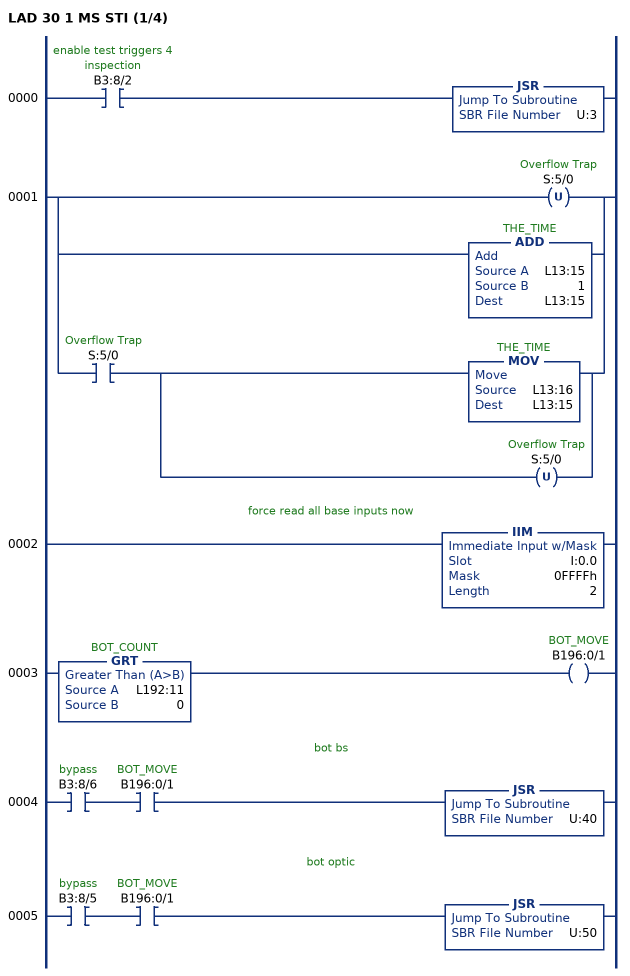
% Rung: 0 %
SOR XIC B3:8/2 JSR U:3 EOR
%   B3:8/2  "enable test triggers 4 inspection" %
% Rung: 1 %
SOR BST OTU S:5/0 NXB ADD L13:15 1 L13:15 NXB XIC S:5/0 BST MOV L13:16 L13:15 NXB OTU S:5/0 BND BND EOR
%   S:5/0  "Overflow Trap" %
%   L13:15  THE_TIME %
%   L13:16  MIN_LONG %
% Rung: 2 %
% force read all base inputs now %
SOR IIM I:0.0 0FFFFh 2 EOR
% Rung: 3 %
SOR GRT L192:11 0 OTE B196:0/1 EOR
%   L192:11  BOT_COUNT %
%   B196:0/1  BOT_MOVE %
% Rung: 4 %
% bot bs %
SOR XIC B3:8/6 XIC B196:0/1 JSR U:40 EOR
%   B3:8/6  "bypass" %
%   B196:0/1  BOT_MOVE %
% Rung: 5 %
% bot optic %
SOR XIC B3:8/5 XIC B196:0/1 JSR U:50 EOR
%   B3:8/5  "bypass" %
%   B196:0/1  BOT_MOVE %

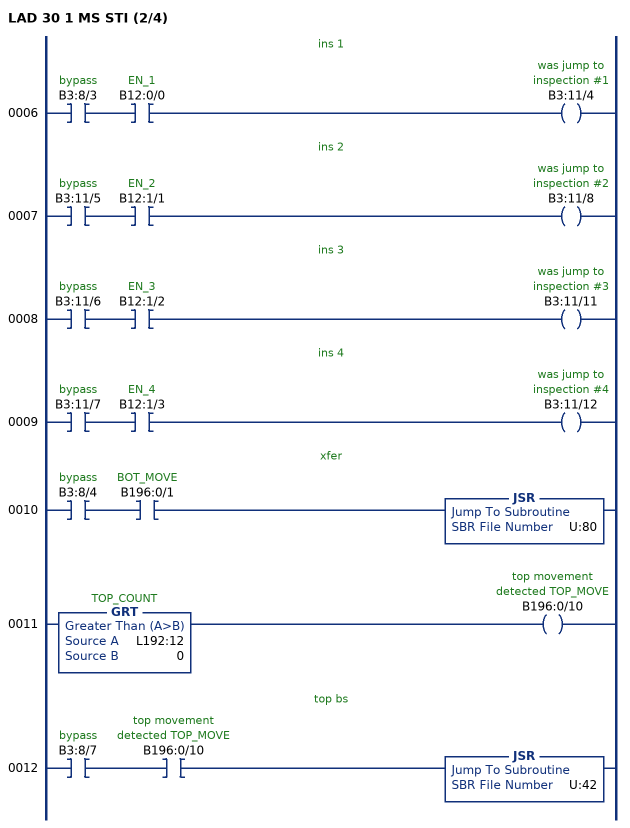
% Rung: 6 %
% ins 1 %
SOR XIC B3:8/3 XIC B12:0/0 OTE B3:11/4 EOR
%   B3:8/3  "bypass" %
%   B12:0/0  EN_1 %
%   B3:11/4  "was jump to inspection #1" %
% Rung: 7 %
% ins 2 %
SOR XIC B3:11/5 XIC B12:1/1 OTE B3:11/8 EOR
%   B3:11/5  "bypass" %
%   B12:1/1  EN_2 %
%   B3:11/8  "was jump to inspection #2" %
% Rung: 8 %
% ins 3 %
SOR XIC B3:11/6 XIC B12:1/2 OTE B3:11/11 EOR
%   B3:11/6  "bypass" %
%   B12:1/2  EN_3 %
%   B3:11/11  "was jump to inspection #3" %
% Rung: 9 %
% ins 4 %
SOR XIC B3:11/7 XIC B12:1/3 OTE B3:11/12 EOR
%   B3:11/7  "bypass" %
%   B12:1/3  EN_4 %
%   B3:11/12  "was jump to inspection #4" %
% Rung: 10 %
% xfer %
SOR XIC B3:8/4 XIC B196:0/1 JSR U:80 EOR
%   B3:8/4  "bypass" %
%   B196:0/1  BOT_MOVE %
% Rung: 11 %
SOR GRT L192:12 0 OTE B196:0/10 EOR
%   L192:12  TOP_COUNT %
%   B196:0/10  TOP_MOVE  "top movement detected" %
% Rung: 12 %
% top bs %
SOR XIC B3:8/7 XIC B196:0/10 JSR U:42 EOR
%   B3:8/7  "bypass" %
%   B196:0/10  TOP_MOVE  "top movement detected" %

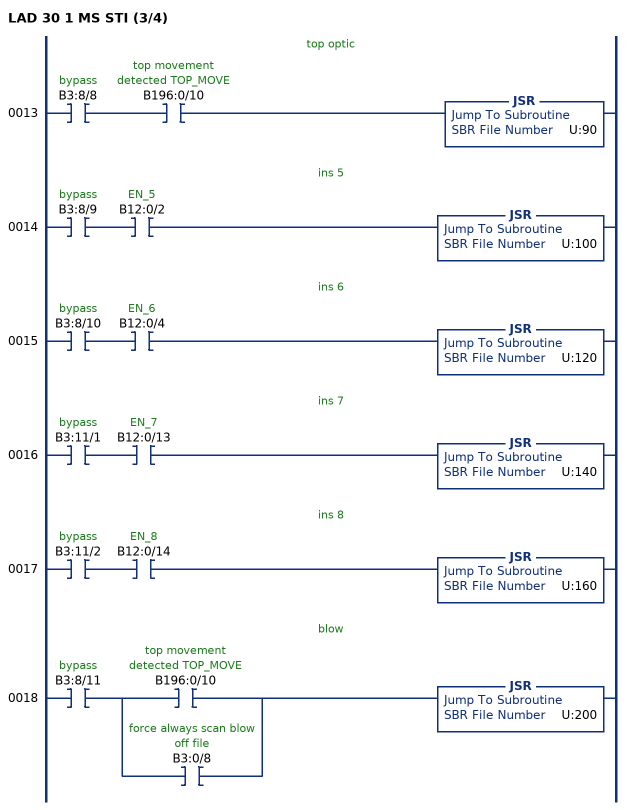
% Rung: 13 %
% top optic %
SOR XIC B3:8/8 XIC B196:0/10 JSR U:90 EOR
%   B3:8/8  "bypass" %
%   B196:0/10  TOP_MOVE  "top movement detected" %
% Rung: 14 %
% ins 5 %
SOR XIC B3:8/9 XIC B12:0/2 JSR U:100 EOR
%   B3:8/9  "bypass" %
%   B12:0/2  EN_5 %
% Rung: 15 %
% ins 6 %
SOR XIC B3:8/10 XIC B12:0/4 JSR U:120 EOR
%   B3:8/10  "bypass" %
%   B12:0/4  EN_6 %
% Rung: 16 %
% ins 7 %
SOR XIC B3:11/1 XIC B12:0/13 JSR U:140 EOR
%   B3:11/1  "bypass" %
%   B12:0/13  EN_7 %
% Rung: 17 %
% ins 8 %
SOR XIC B3:11/2 XIC B12:0/14 JSR U:160 EOR
%   B3:11/2  "bypass" %
%   B12:0/14  EN_8 %
% Rung: 18 %
% blow %
SOR XIC B3:8/11 BST XIC B196:0/10 NXB XIC B3:0/8 BND JSR U:200 EOR
%   B3:8/11  "bypass" %
%   B196:0/10  TOP_MOVE  "top movement detected" %
%   B3:0/8  "force always scan blow off file" %

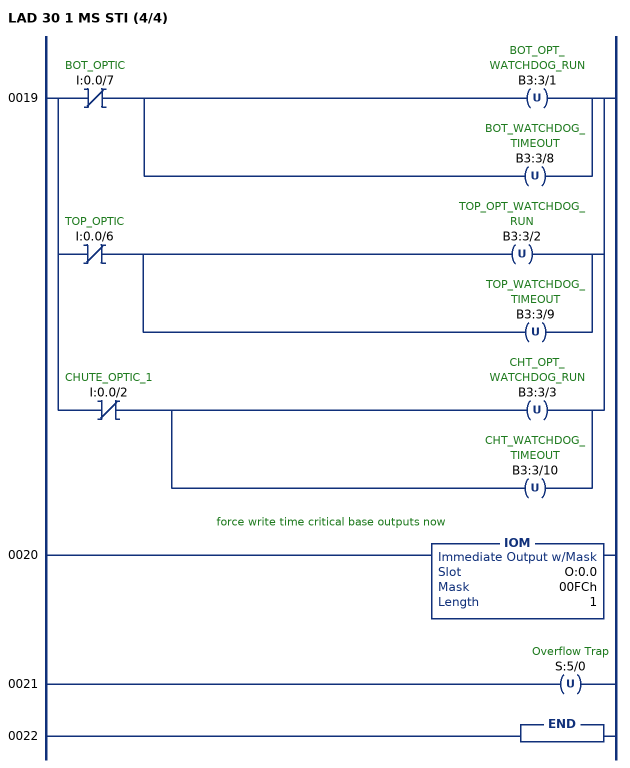
% Rung: 19 %
SOR BST XIO I:0.0/7 BST OTU B3:3/1 NXB OTU B3:3/8 BND NXB XIO I:0.0/6 BST OTU B3:3/2 NXB OTU B3:3/9 BND NXB XIO I:0.0/2 BST OTU B3:3/3 NXB OTU B3:3/10 BND BND EOR
%   I:0.0/7  BOT_OPTIC %
%   B3:3/1  BOT_OPT_WATCHDOG_RUN %
%   B3:3/8  BOT_WATCHDOG_TIMEOUT %
%   I:0.0/6  TOP_OPTIC %
%   B3:3/2  TOP_OPT_WATCHDOG_RUN %
%   B3:3/9  TOP_WATCHDOG_TIMEOUT %
%   I:0.0/2  CHUTE_OPTIC_1 %
%   B3:3/3  CHT_OPT_WATCHDOG_RUN %
%   B3:3/10  CHT_WATCHDOG_TIMEOUT %
% Rung: 20 %
% force write time critical base outputs now %
SOR IOM O:0.0 00FCh 1 EOR
% Rung: 21 %
SOR OTU S:5/0 EOR
%   S:5/0  "Overflow Trap" %
% Rung: 22 %
SOR END EOR

LADDER 40 "SHIFT BOT"
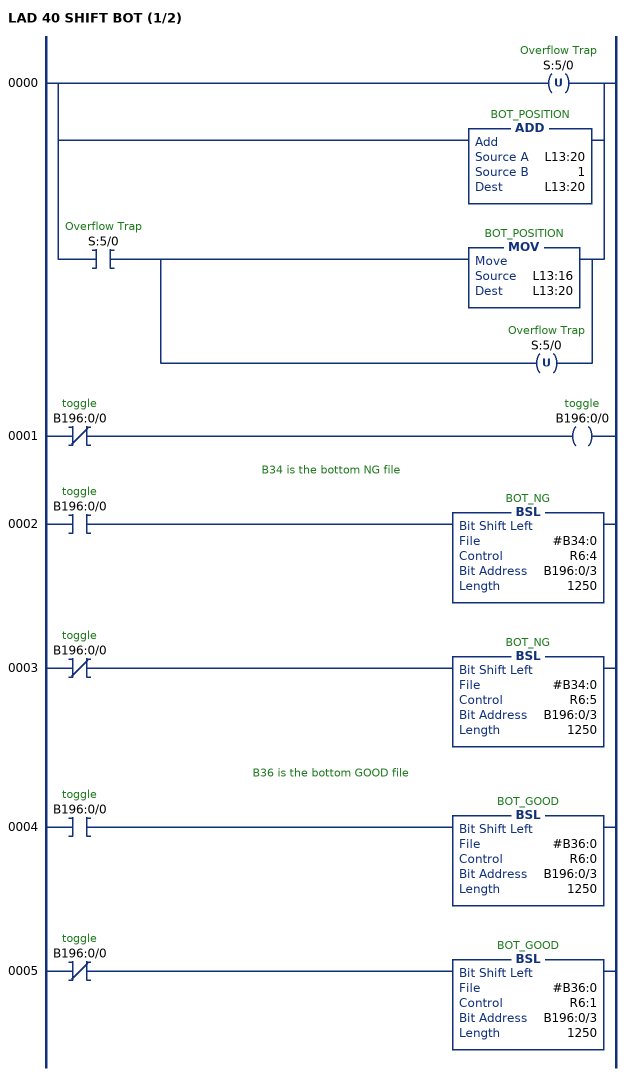
% Rung: 0 %
SOR BST OTU S:5/0 NXB ADD L13:20 1 L13:20 NXB XIC S:5/0 BST MOV L13:16 L13:20 NXB OTU S:5/0 BND BND EOR
%   S:5/0  "Overflow Trap" %
%   L13:20  BOT_POSITION %
%   L13:16  MIN_LONG %
% Rung: 1 %
SOR XIO B196:0/0 OTE B196:0/0 EOR
%   B196:0/0  "toggle" %
% Rung: 2 %
% B34 is the bottom NG file %
SOR XIC B196:0/0 BSL #B34:0 R6:4 B196:0/3 1250 EOR
%   B196:0/0  "toggle" %
%   B34:0  BOT_NG %
%   B196:0/3  OFF %
% Rung: 3 %
SOR XIO B196:0/0 BSL #B34:0 R6:5 B196:0/3 1250 EOR
%   B196:0/0  "toggle" %
%   B34:0  BOT_NG %
%   B196:0/3  OFF %
% Rung: 4 %
% B36 is the bottom GOOD file %
SOR XIC B196:0/0 BSL #B36:0 R6:0 B196:0/3 1250 EOR
%   B196:0/0  "toggle" %
%   B36:0  BOT_GOOD %
%   B196:0/3  OFF %
% Rung: 5 %
SOR XIO B196:0/0 BSL #B36:0 R6:1 B196:0/3 1250 EOR
%   B196:0/0  "toggle" %
%   B36:0  BOT_GOOD %
%   B196:0/3  OFF %

